// TIA Portal V20 export
FUNCTION "Service_Filling" : Void   // FC23, FBD
TITLE = Service
{ S7_Optimized_Access := 'TRUE' }
AUTHOR : Siemens AG
FAMILY : ServiceControl
VERSION : 1.0
// stored: SetENOAutomatically false
   VAR_TEMP
      StartingState : Bool;
      CompletingState : Bool;
      PausingState : Bool;
      HoldingState : Bool;
      AbortingState : Bool;
      StoppingState : Bool;
      ExecuteState : Bool;
      State : "Service_States";
   END_VAR
BEGIN

REGION Network 1: Prepare feedback
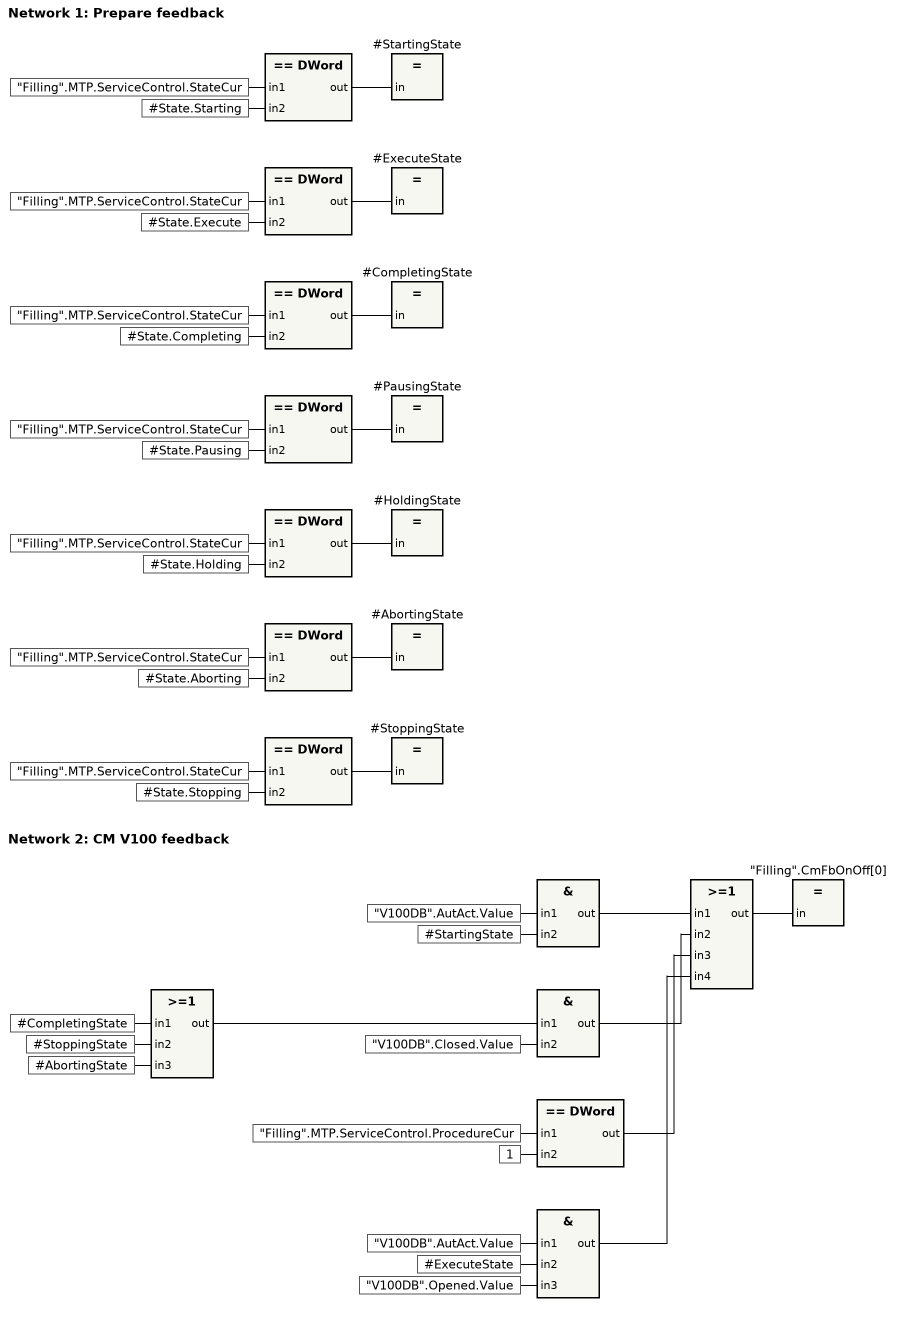
   #StartingState := "Filling".MTP.ServiceControl.StateCur = #State.Starting;
   #ExecuteState := "Filling".MTP.ServiceControl.StateCur = #State.Execute;
   #CompletingState := "Filling".MTP.ServiceControl.StateCur = #State.Completing;
   #PausingState := "Filling".MTP.ServiceControl.StateCur = #State.Pausing;
   #HoldingState := "Filling".MTP.ServiceControl.StateCur = #State.Holding;
   #AbortingState := "Filling".MTP.ServiceControl.StateCur = #State.Aborting;
   #StoppingState := "Filling".MTP.ServiceControl.StateCur = #State.Stopping;
END_REGION

REGION Network 2: CM V100 feedback
   "Filling".CmFbOnOff[0] := ("V100DB".AutAct.Value AND #StartingState) OR ((#CompletingState OR #StoppingState OR #AbortingState) AND "V100DB".Closed.Value) OR ("Filling".MTP.ServiceControl.ProcedureCur = 1) OR ("V100DB".AutAct.Value AND #ExecuteState AND "V100DB".Opened.Value);
END_REGION

REGION Network 3: CM V101 feedback
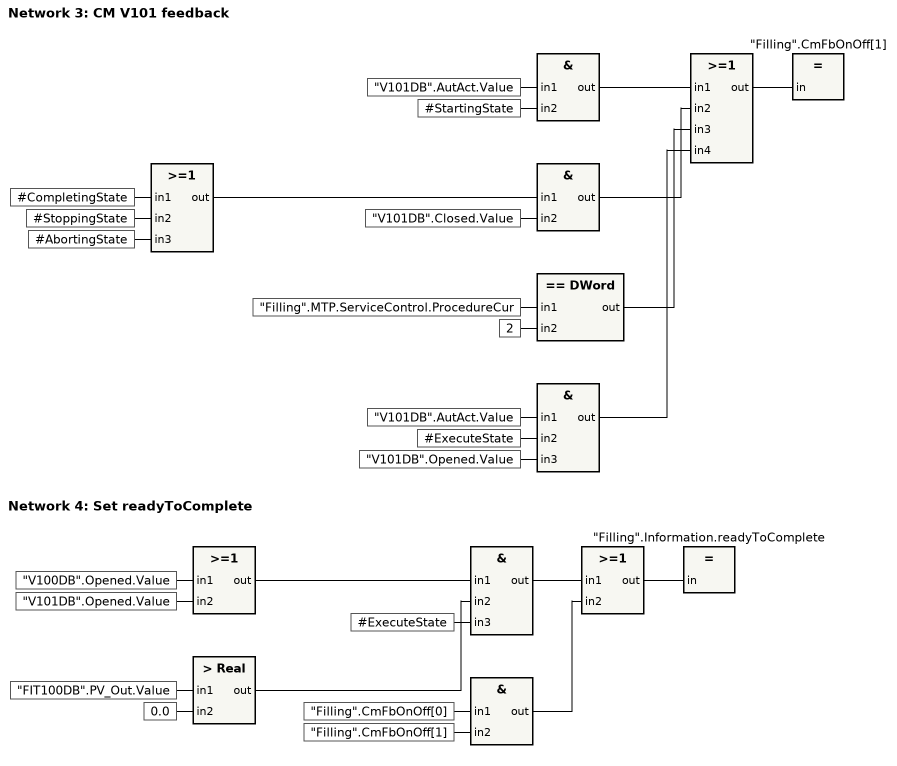
   "Filling".CmFbOnOff[1] := ("V101DB".AutAct.Value AND #StartingState) OR ((#CompletingState OR #StoppingState OR #AbortingState) AND "V101DB".Closed.Value) OR ("Filling".MTP.ServiceControl.ProcedureCur = 2) OR ("V101DB".AutAct.Value AND #ExecuteState AND "V101DB".Opened.Value);
END_REGION

REGION Network 4: Set readyToComplete
   "Filling".Information.readyToComplete := (("V100DB".Opened.Value OR "V101DB".Opened.Value) AND ("FIT100DB".PV_Out.Value > 0.0) AND #ExecuteState) OR ("Filling".CmFbOnOff[0] AND "Filling".CmFbOnOff[1]);
END_REGION

REGION Network 5: Service
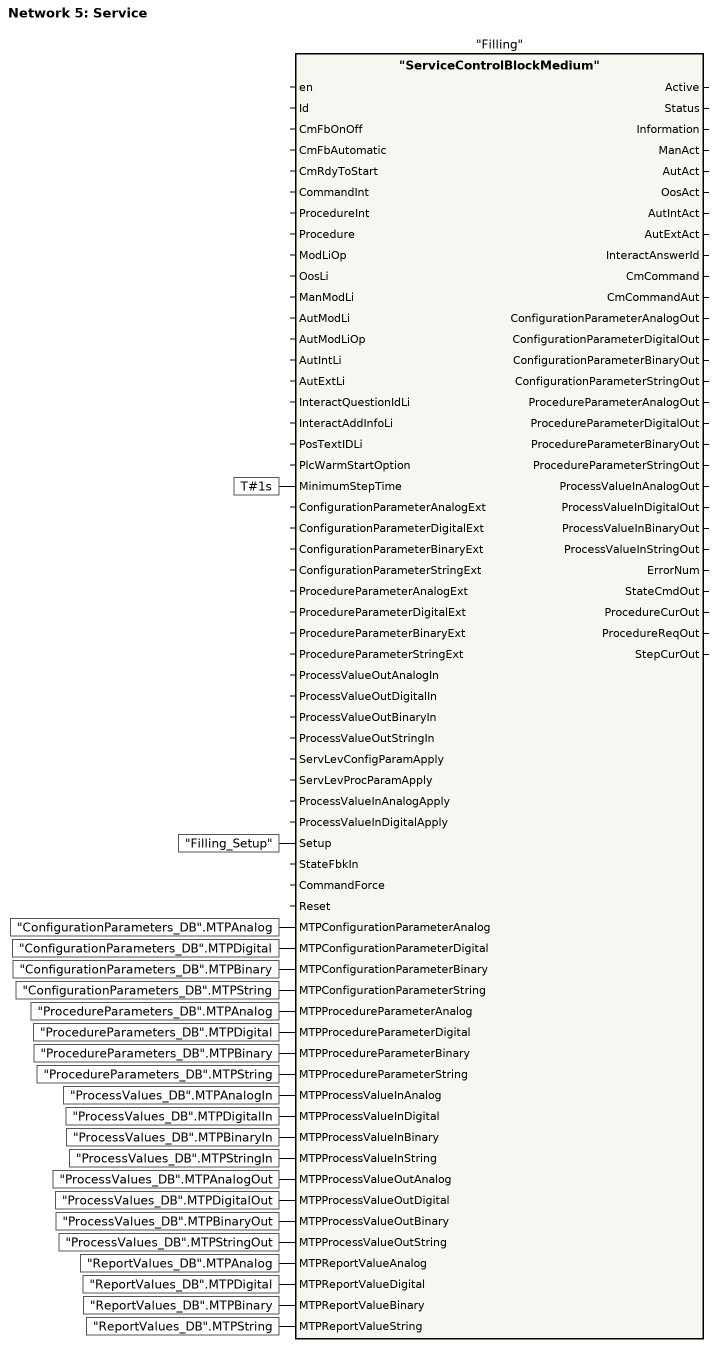
   "Filling"(MinimumStepTime := T#1s,   // "ServiceControlBlockMedium"
             Setup := "Filling_Setup",
             MTPConfigurationParameterAnalog := "ConfigurationParameters_DB".MTPAnalog,
             MTPConfigurationParameterDigital := "ConfigurationParameters_DB".MTPDigital,
             MTPConfigurationParameterBinary := "ConfigurationParameters_DB".MTPBinary,
             MTPConfigurationParameterString := "ConfigurationParameters_DB".MTPString,
             MTPProcedureParameterAnalog := "ProcedureParameters_DB".MTPAnalog,
             MTPProcedureParameterDigital := "ProcedureParameters_DB".MTPDigital,
             MTPProcedureParameterBinary := "ProcedureParameters_DB".MTPBinary,
             MTPProcedureParameterString := "ProcedureParameters_DB".MTPString,
             MTPProcessValueInAnalog := "ProcessValues_DB".MTPAnalogIn,
             MTPProcessValueInDigital := "ProcessValues_DB".MTPDigitalIn,
             MTPProcessValueInBinary := "ProcessValues_DB".MTPBinaryIn,
             MTPProcessValueInString := "ProcessValues_DB".MTPStringIn,
             MTPProcessValueOutAnalog := "ProcessValues_DB".MTPAnalogOut,
             MTPProcessValueOutDigital := "ProcessValues_DB".MTPDigitalOut,
             MTPProcessValueOutBinary := "ProcessValues_DB".MTPBinaryOut,
             MTPProcessValueOutString := "ProcessValues_DB".MTPStringOut,
             MTPReportValueAnalog := "ReportValues_DB".MTPAnalog,
             MTPReportValueDigital := "ReportValues_DB".MTPDigital,
             MTPReportValueBinary := "ReportValues_DB".MTPBinary,
             MTPReportValueString := "ReportValues_DB".MTPString);
END_REGION

REGION Network 6: Service HMI
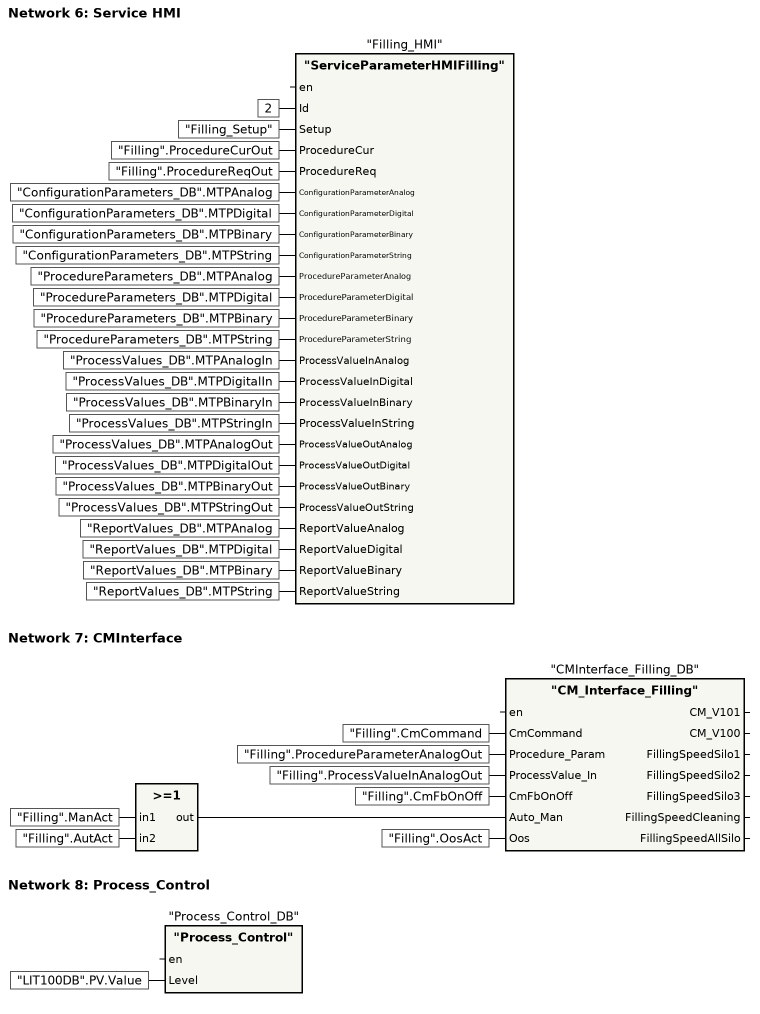
   "Filling_HMI"(Id := 2,   // "ServiceParameterHMIFilling"
                 Setup := "Filling_Setup",
                 ProcedureCur := "Filling".ProcedureCurOut,
                 ProcedureReq := "Filling".ProcedureReqOut,
                 ConfigurationParameterAnalog := "ConfigurationParameters_DB".MTPAnalog,
                 ConfigurationParameterDigital := "ConfigurationParameters_DB".MTPDigital,
                 ConfigurationParameterBinary := "ConfigurationParameters_DB".MTPBinary,
                 ConfigurationParameterString := "ConfigurationParameters_DB".MTPString,
                 ProcedureParameterAnalog := "ProcedureParameters_DB".MTPAnalog,
                 ProcedureParameterDigital := "ProcedureParameters_DB".MTPDigital,
                 ProcedureParameterBinary := "ProcedureParameters_DB".MTPBinary,
                 ProcedureParameterString := "ProcedureParameters_DB".MTPString,
                 ProcessValueInAnalog := "ProcessValues_DB".MTPAnalogIn,
                 ProcessValueInDigital := "ProcessValues_DB".MTPDigitalIn,
                 ProcessValueInBinary := "ProcessValues_DB".MTPBinaryIn,
                 ProcessValueInString := "ProcessValues_DB".MTPStringIn,
                 ProcessValueOutAnalog := "ProcessValues_DB".MTPAnalogOut,
                 ProcessValueOutDigital := "ProcessValues_DB".MTPDigitalOut,
                 ProcessValueOutBinary := "ProcessValues_DB".MTPBinaryOut,
                 ProcessValueOutString := "ProcessValues_DB".MTPStringOut,
                 ReportValueAnalog := "ReportValues_DB".MTPAnalog,
                 ReportValueDigital := "ReportValues_DB".MTPDigital,
                 ReportValueBinary := "ReportValues_DB".MTPBinary,
                 ReportValueString := "ReportValues_DB".MTPString);
END_REGION

REGION Network 7: CMInterface
   "CMInterface_Filling_DB"(CmCommand := "Filling".CmCommand,   // "CM_Interface_Filling"
                           Procedure_Param := "Filling".ProcedureParameterAnalogOut,
                           ProcessValue_In := "Filling".ProcessValueInAnalogOut,
                           CmFbOnOff := "Filling".CmFbOnOff,
                           Auto_Man := "Filling".ManAct OR "Filling".AutAct,
                           Oos := "Filling".OosAct);
END_REGION

REGION Network 8: Process_Control
   "Process_Control_DB"(Level := "LIT100DB".PV.Value);   // "Process_Control"
END_REGION

REGION Network 9: Block pause and hold state
END_REGION

REGION Network 10: Report values and Process Value Out
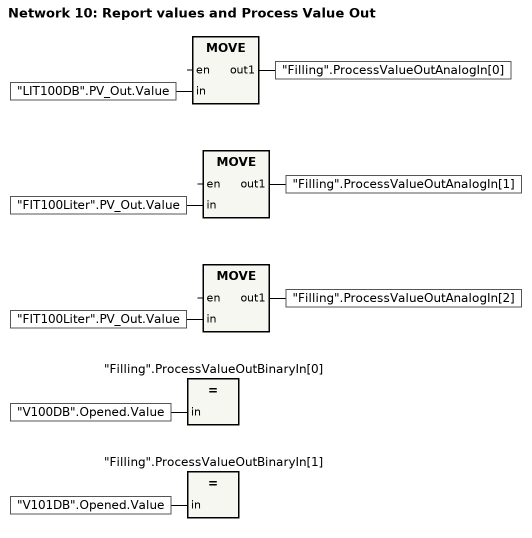
   "Filling".ProcessValueOutAnalogIn[0] := "LIT100DB".PV_Out.Value;
   "Filling".ProcessValueOutAnalogIn[1] := "FIT100Liter".PV_Out.Value;
   "Filling".ProcessValueOutAnalogIn[2] := "FIT100Liter".PV_Out.Value;
   "Filling".ProcessValueOutBinaryIn[0] := "V100DB".Opened.Value;
   "Filling".ProcessValueOutBinaryIn[1] := "V101DB".Opened.Value;
END_REGION
END_FUNCTION
